(* Logix 5000 project; controller STAT 1756-L72 rev 20.12; software revision 20.04; part 32 of 34 *)
(* tags used below, declared in another part *)
   B3 : DINT[50];
   F8 : REAL[200];
   I2_000_Bit12 : ALIAS FOR stock:2:I.Point_12;   // chaudière wanson0= on 1= off
   I2_000_Bit13 : ALIAS FOR stock:2:I.Point_13;   // chaudière colmatageLigne 30= on 1= off
   I2_001_Bit00 : ALIAS FOR stock:2:I.Point_16;   // NAOHL1 VA4FC O
   I2_001_Bit01 : ALIAS FOR stock:2:I.Point_17;   // NAOHL1 VA4FC F
   I2_001_Bit02 : ALIAS FOR stock:2:I.Point_18;   // NAOHL2 VA4FC O
   I2_001_Bit03 : ALIAS FOR stock:2:I.Point_19;   // NAOHL2 VA4FC O
   I2_001_Bit06 : ALIAS FOR stock:2:I.Point_22;   // pulse debitmetreacide 0.2 l
   I2_001_Bit07 : ALIAS FOR stock:2:I.Point_23;   // pulse eau in tourL1 &2
   I2_001_Bit15 : ALIAS FOR stock:2:I.Point_31;   // pulse 0.1L passé
   I5_000 : ALIAS FOR stock:5:I.Channel_0_Data;
   N20 : DINT[100];
   N7 : DINT[255];
   O3_000_Bit02 : ALIAS FOR stock:3:O.Point_2;   // pompe acide
   O3_000_Bit08 : ALIAS FOR stock:3:O.Point_8;   // vanne soude
   S_V_NAOH : BOOL;
   T4 : TIMER[50];
   dmd_h2so4_ibt_ok : BOOL;
   dmd_soude_ibt_ok : BOOL;
   h2so4_ibt_finit : BOOL;
   ibt_level_soude_plein : BOOL;
   L1_stat : DINT[20];
   L2_STAT : DINT[20];
   L3_STAT : DINT[20];
   lancystock2 : DINT;
   N : INT[255];
   N12 : DINT[230];
   ons12 : BOOL;
   ONS13 : BOOL;
   ONS3 : BOOL;
   ONS4 : BOOL;
   ONS5 : BOOL;
   s_acide_ibt_passe : REAL;
   s_bp_start_h2so4_ibt : BOOL;
   s_bp_stop_acide_ibt : BOOL;
   s_bp_stop_soude_ibt : BOOL;
   s_dmd_acid_ibt : DINT;
   s_h2so4_ibt : BOOL;
   S_naoh_ibt : BOOL;
   S_naoh_ibt_passe : REAL;
   S_stock_v_h2so4_f : BOOL;
   S_stock_v_h2so4_o : BOOL;
   S_stock_v_naoh_o : BOOL;
   stat_L1 : DINT[20];
   STAT_L2 : DINT[20];
   STAT_L3 : DINT[20];
   stocklancy1 : DINT;
   stocklancy2 : DINT;
   stocklancy3 : DINT;
   tot_gaz_chaud_iwts_L123 : DINT;   // 19/1/15 13h45
   tot_gaz_chaud_L3 : DINT;   // debut le 16/1/15 à 11h30
   tot_gaz_chaud_wanson : DINT;   // 19/1/15 13h45
   tot_h2so4_stat : REAL;
(* stock, continued *)

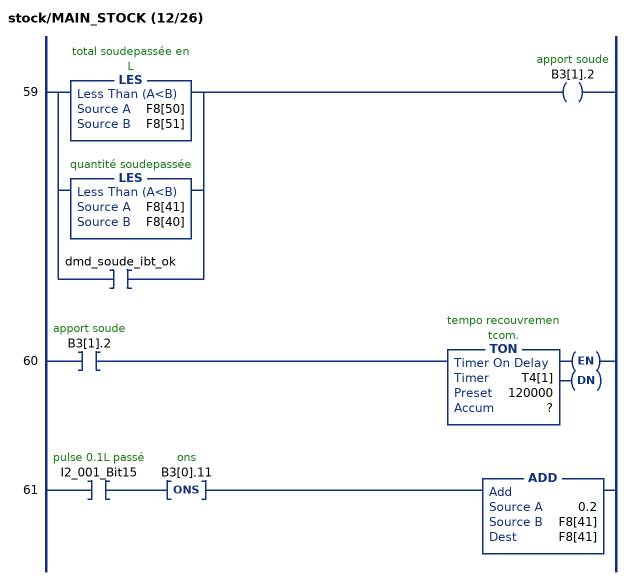
   [picture p650: stock/MAIN_STOCK rungs 59-61]
   59: [LES(F8[50],F8[51]) ,LES(F8[41],F8[40]) ,XIC(dmd_soude_ibt_ok) ]OTE(B3[1].2);
   60: XIC(B3[1].2)TON(T4[1],?,?);
   61: XIC(I2_001_Bit15)ONS(B3[0].11)ADD(0.2,F8[41],F8[41]);
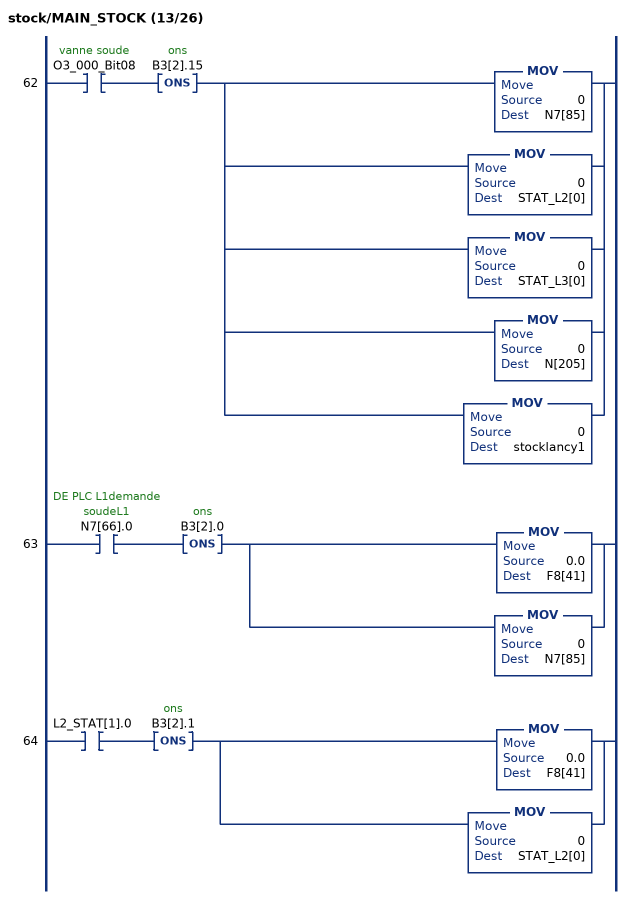
   62: XIC(O3_000_Bit08)ONS(B3[2].15)[MOV(0,N7[85]) ,MOV(0,STAT_L2[0]) ,MOV(0,STAT_L3[0]) ,MOV(0,N[205]) ,MOV(0,stocklancy1) ];
   63: XIC(N7[66].0)ONS(B3[2].0)[MOV(0.0,F8[41]) ,MOV(0,N7[85]) ];
   64: XIC(L2_STAT[1].0)ONS(B3[2].1)[MOV(0.0,F8[41]) ,MOV(0,STAT_L2[0]) ];
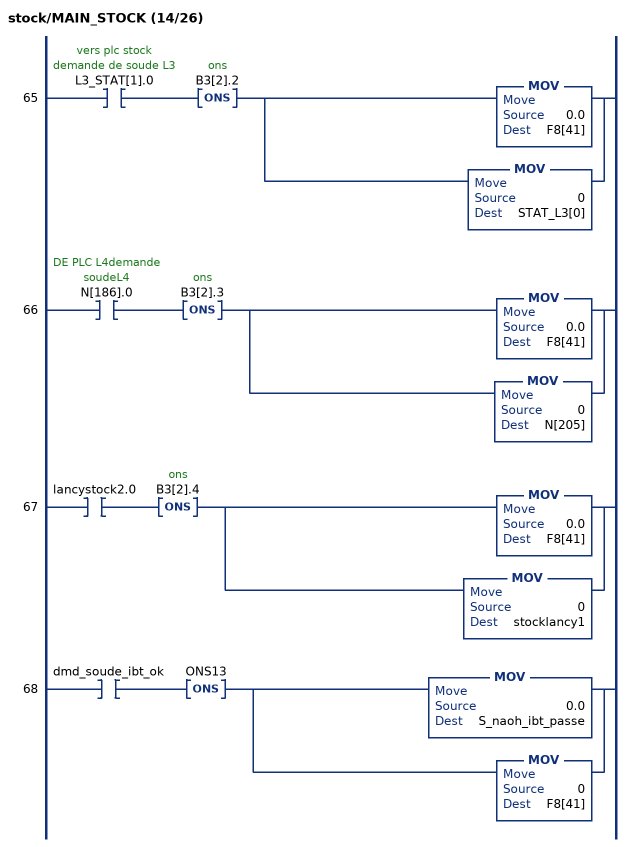
   65: XIC(L3_STAT[1].0)ONS(B3[2].2)[MOV(0.0,F8[41]) ,MOV(0,STAT_L3[0]) ];
   66: XIC(N[186].0)ONS(B3[2].3)[MOV(0.0,F8[41]) ,MOV(0,N[205]) ];
   67: XIC(lancystock2.0)ONS(B3[2].4)[MOV(0.0,F8[41]) ,MOV(0,stocklancy1) ];
   68: XIC(dmd_soude_ibt_ok)ONS(ONS13)[MOV(0.0,S_naoh_ibt_passe) ,MOV(0,F8[41]) ];
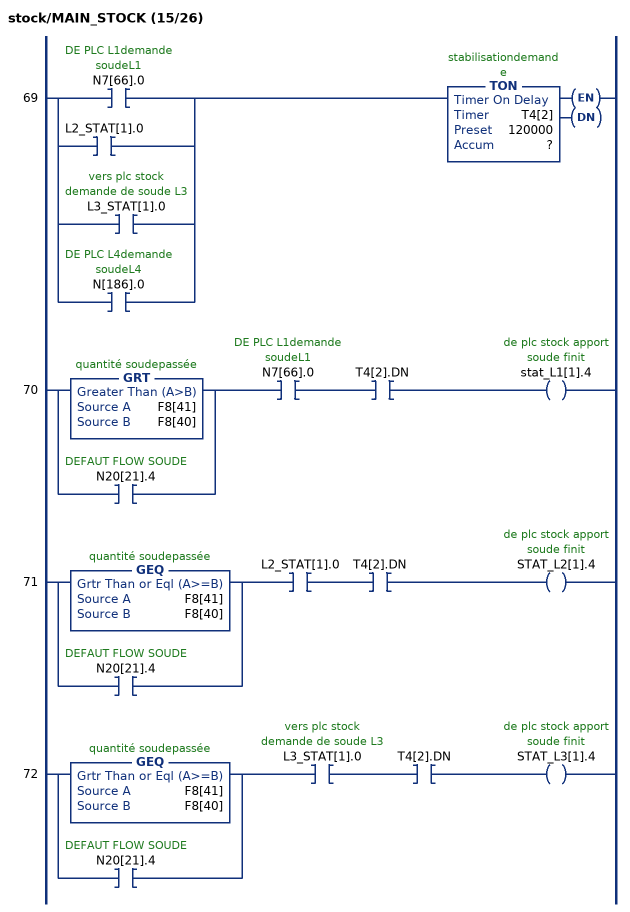
   69: [XIC(N7[66].0) ,XIC(L2_STAT[1].0) ,XIC(L3_STAT[1].0) ,XIC(N[186].0) ]TON(T4[2],?,?);
   70: [GRT(F8[41],F8[40]) ,XIC(N20[21].4) ]XIC(N7[66].0)XIC(T4[2].DN)OTE(stat_L1[1].4);
   71: [GEQ(F8[41],F8[40]) ,XIC(N20[21].4) ]XIC(L2_STAT[1].0)XIC(T4[2].DN)OTE(STAT_L2[1].4);
   72: [GEQ(F8[41],F8[40]) ,XIC(N20[21].4) ]XIC(L3_STAT[1].0)XIC(T4[2].DN)OTE(STAT_L3[1].4);
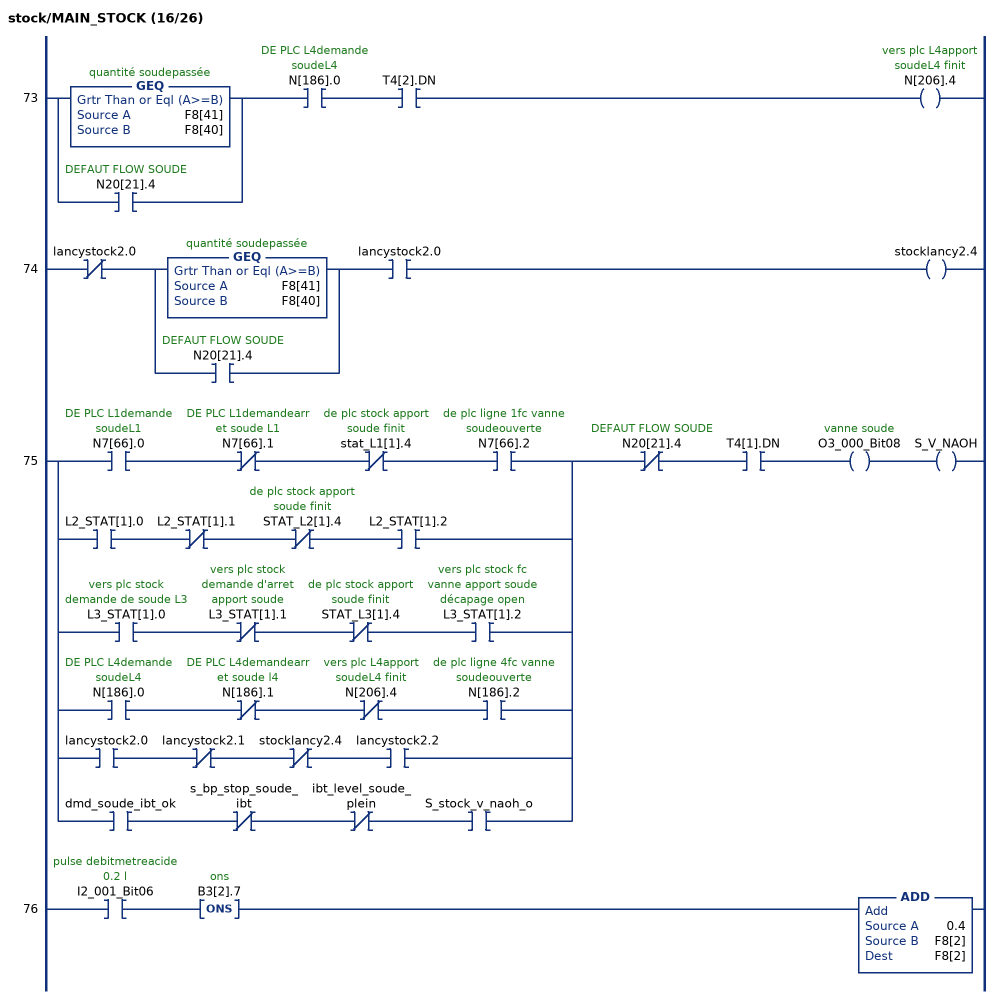
   73: [GEQ(F8[41],F8[40]) ,XIC(N20[21].4) ]XIC(N[186].0)XIC(T4[2].DN)OTE(N[206].4);
   74: XIO(lancystock2.0)[GEQ(F8[41],F8[40]) ,XIC(N20[21].4) ]XIC(lancystock2.0)OTE(stocklancy2.4);
   75: [XIC(N7[66].0) XIO(N7[66].1) XIO(stat_L1[1].4) XIC(N7[66].2) ,XIC(L2_STAT[1].0) XIO(L2_STAT[1].1) XIO(STAT_L2[1].4) XIC(L2_STAT[1].2) ,XIC(L3_STAT[1].0) XIO(L3_STAT[1].1) XIO(STAT_L3[1].4) XIC(L3_STAT[1].2) ,XIC(N[186].0) XIO(N[186].1) XIO(N[206].4) XIC(N[186].2) ,XIC(lancystock2.0) XIO(lancystock2.1) XIO(stocklancy2.4) XIC(lancystock2.2) ,XIC(dmd_soude_ibt_ok) XIO(s_bp_stop_soude_ibt) XIO(ibt_level_soude_plein) XIC(S_stock_v_naoh_o) ]XIO(N20[21].4)XIC(T4[1].DN)OTE(O3_000_Bit08)OTE(S_V_NAOH);
   76: XIC(I2_001_Bit06)ONS(B3[2].7)ADD(0.4,F8[2],F8[2]);
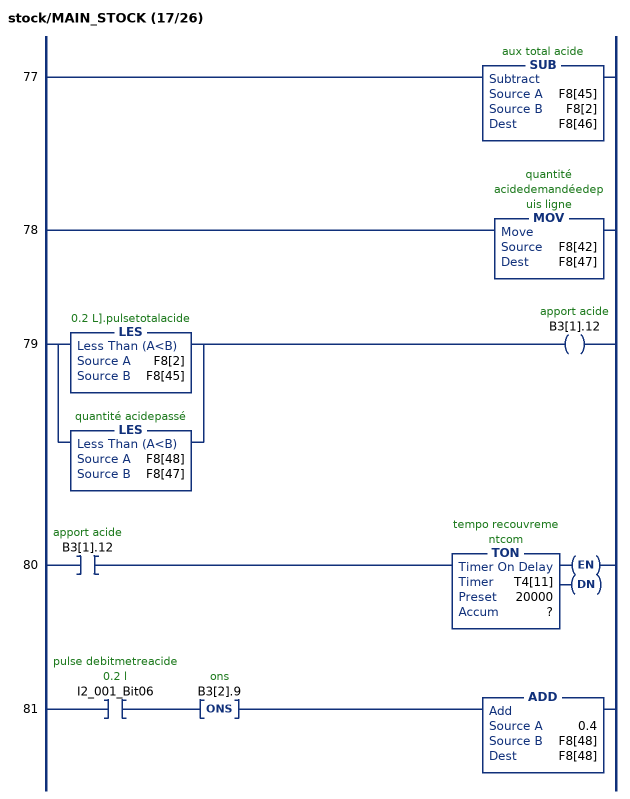
   77: SUB(F8[45],F8[2],F8[46]);
   78: MOV(F8[42],F8[47]);
   79: [LES(F8[2],F8[45]) ,LES(F8[48],F8[47]) ]OTE(B3[1].12);
   80: XIC(B3[1].12)TON(T4[11],?,?);
   81: XIC(I2_001_Bit06)ONS(B3[2].9)ADD(0.4,F8[48],F8[48]);
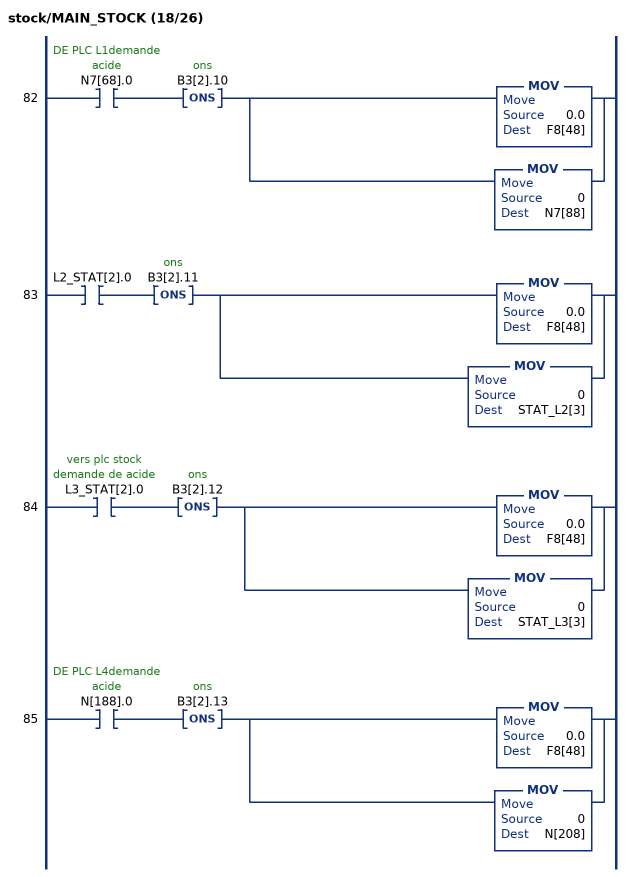
   82: XIC(N7[68].0)ONS(B3[2].10)[MOV(0.0,F8[48]) ,MOV(0,N7[88]) ];
   83: XIC(L2_STAT[2].0)ONS(B3[2].11)[MOV(0.0,F8[48]) ,MOV(0,STAT_L2[3]) ];
   84: XIC(L3_STAT[2].0)ONS(B3[2].12)[MOV(0.0,F8[48]) ,MOV(0,STAT_L3[3]) ];
   85: XIC(N[188].0)ONS(B3[2].13)[MOV(0.0,F8[48]) ,MOV(0,N[208]) ];
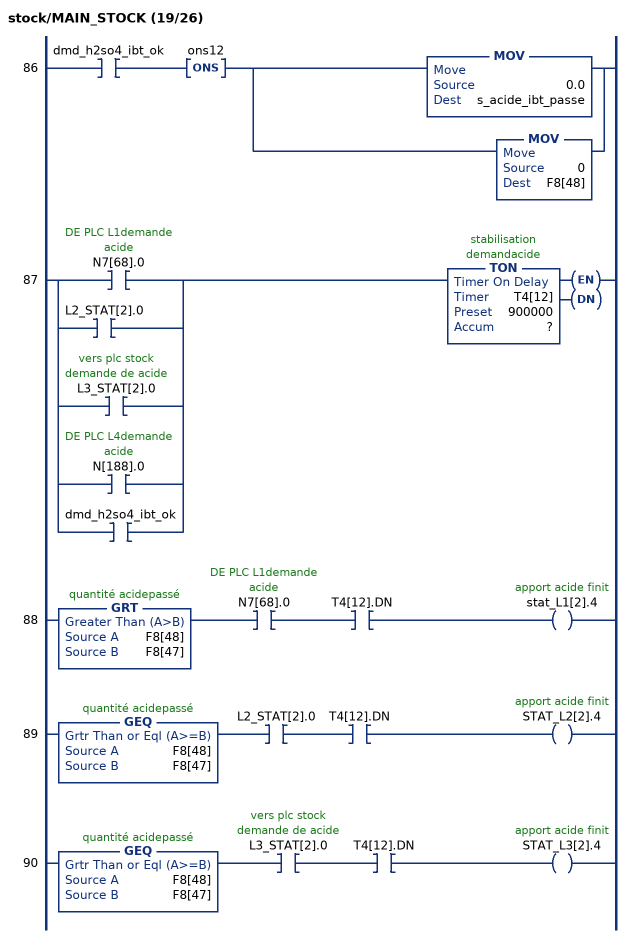
   86: XIC(dmd_h2so4_ibt_ok)ONS(ons12)[MOV(0.0,s_acide_ibt_passe) ,MOV(0,F8[48]) ];
   87: [XIC(N7[68].0) ,XIC(L2_STAT[2].0) ,XIC(L3_STAT[2].0) ,XIC(N[188].0) ,XIC(dmd_h2so4_ibt_ok) ]TON(T4[12],?,?);
   88: GRT(F8[48],F8[47])XIC(N7[68].0)XIC(T4[12].DN)OTE(stat_L1[2].4);
   89: GEQ(F8[48],F8[47])XIC(L2_STAT[2].0)XIC(T4[12].DN)OTE(STAT_L2[2].4);
   90: GEQ(F8[48],F8[47])XIC(L3_STAT[2].0)XIC(T4[12].DN)OTE(STAT_L3[2].4);
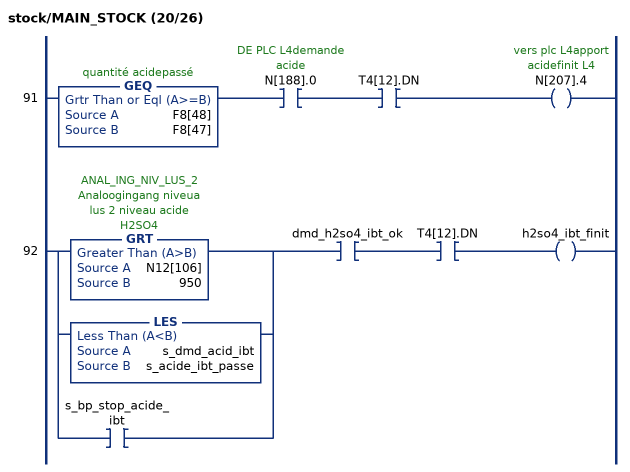
   91: GEQ(F8[48],F8[47])XIC(N[188].0)XIC(T4[12].DN)OTE(N[207].4);
   92: [GRT(N12[106],950) ,LES(s_dmd_acid_ibt,s_acide_ibt_passe) ,XIC(s_bp_stop_acide_ibt) ]XIC(dmd_h2so4_ibt_ok)XIC(T4[12].DN)OTE(h2so4_ibt_finit);
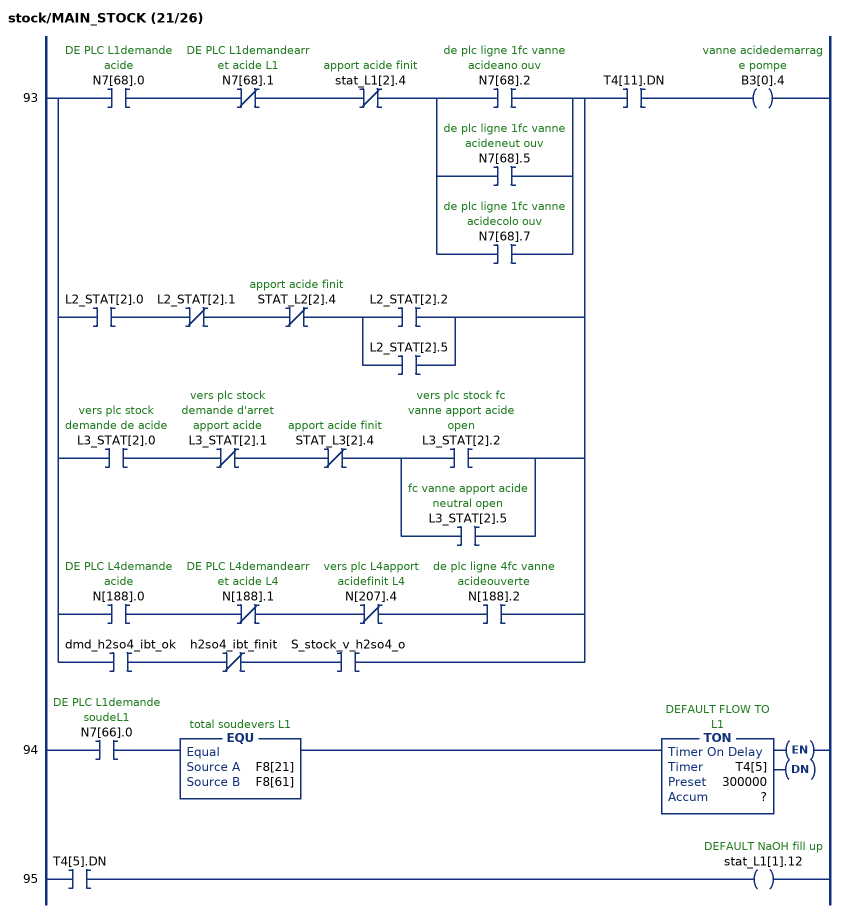
   93: [XIC(N7[68].0) XIO(N7[68].1) XIO(stat_L1[2].4) [XIC(N7[68].2) ,XIC(N7[68].5) ,XIC(N7[68].7) ] ,XIC(L2_STAT[2].0) XIO(L2_STAT[2].1) XIO(STAT_L2[2].4) [XIC(L2_STAT[2].2) ,XIC(L2_STAT[2].5) ] ,XIC(L3_STAT[2].0) XIO(L3_STAT[2].1) XIO(STAT_L3[2].4) [XIC(L3_STAT[2].2) ,XIC(L3_STAT[2].5) ] ,XIC(N[188].0) XIO(N[188].1) XIO(N[207].4) XIC(N[188].2) ,XIC(dmd_h2so4_ibt_ok) XIO(h2so4_ibt_finit) XIC(S_stock_v_h2so4_o) ]XIC(T4[11].DN)OTE(B3[0].4);
   94: XIC(N7[66].0)EQU(F8[21],F8[61])TON(T4[5],?,?);
   95: XIC(T4[5].DN)OTE(stat_L1[1].12);
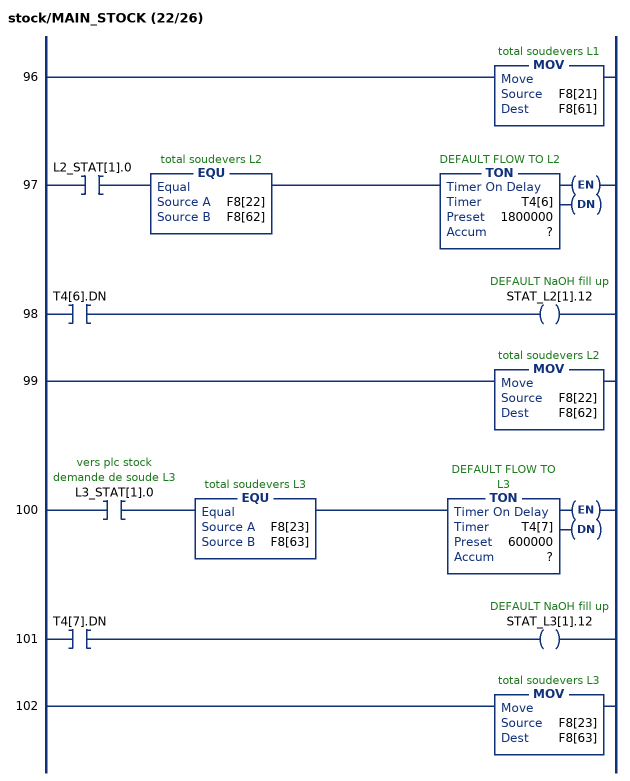
   96: MOV(F8[21],F8[61]);
   97: XIC(L2_STAT[1].0)EQU(F8[22],F8[62])TON(T4[6],?,?);
   98: XIC(T4[6].DN)OTE(STAT_L2[1].12);
   99: MOV(F8[22],F8[62]);
   100: XIC(L3_STAT[1].0)EQU(F8[23],F8[63])TON(T4[7],?,?);
   101: XIC(T4[7].DN)OTE(STAT_L3[1].12);
   102: MOV(F8[23],F8[63]);
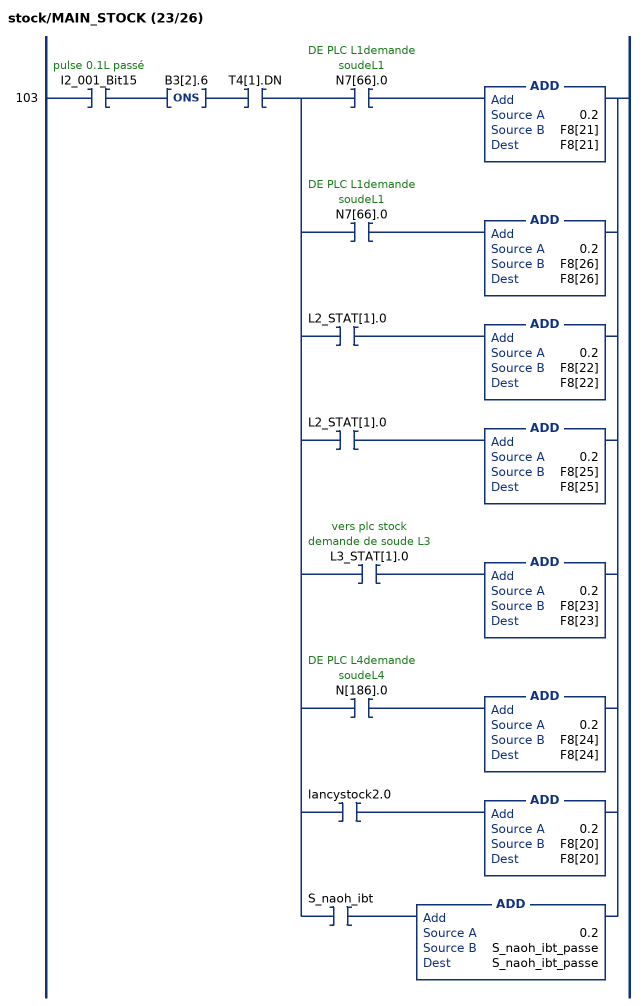
   103: XIC(I2_001_Bit15)ONS(B3[2].6)XIC(T4[1].DN)[XIC(N7[66].0) ADD(0.2,F8[21],F8[21]) ,XIC(N7[66].0) ADD(0.2,F8[26],F8[26]) ,XIC(L2_STAT[1].0) ADD(0.2,F8[22],F8[22]) ,XIC(L2_STAT[1].0) ADD(0.2,F8[25],F8[25]) ,XIC(L3_STAT[1].0) ADD(0.2,F8[23],F8[23]) ,XIC(N[186].0) ADD(0.2,F8[24],F8[24]) ,XIC(lancystock2.0) ADD(0.2,F8[20],F8[20]) ,XIC(S_naoh_ibt) ADD(0.2,S_naoh_ibt_passe,S_naoh_ibt_passe) ];
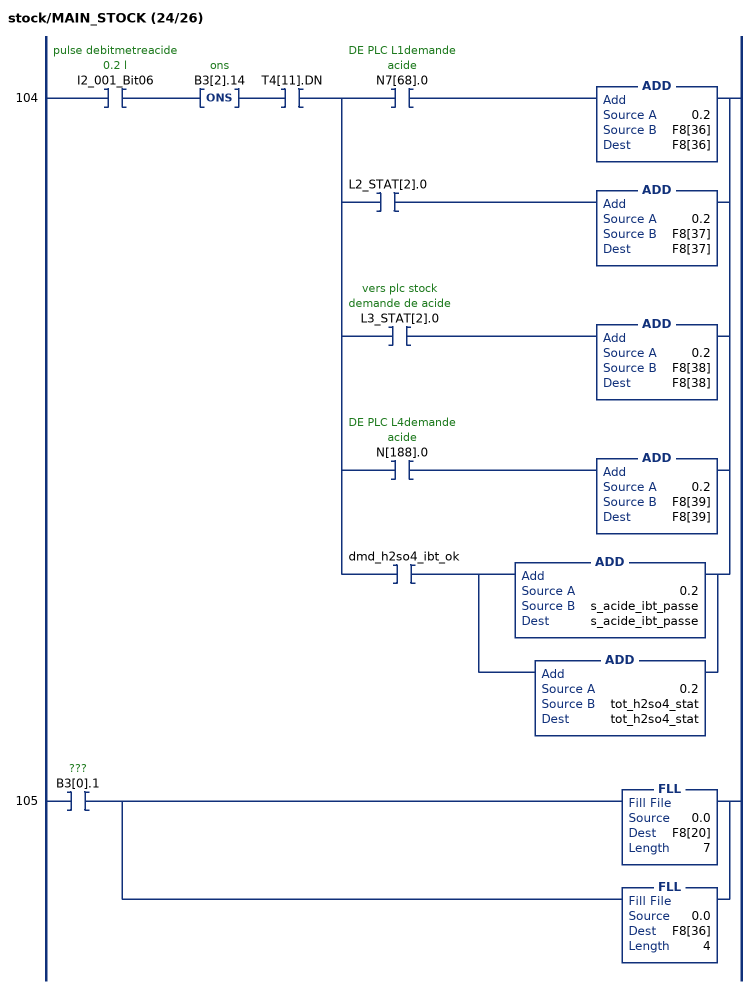
   104: XIC(I2_001_Bit06)ONS(B3[2].14)XIC(T4[11].DN)[XIC(N7[68].0) ADD(0.2,F8[36],F8[36]) ,XIC(L2_STAT[2].0) ADD(0.2,F8[37],F8[37]) ,XIC(L3_STAT[2].0) ADD(0.2,F8[38],F8[38]) ,XIC(N[188].0) ADD(0.2,F8[39],F8[39]) ,XIC(dmd_h2so4_ibt_ok) [ADD(0.2,s_acide_ibt_passe,s_acide_ibt_passe) ,ADD(0.2,tot_h2so4_stat,tot_h2so4_stat) ] ];
   105: XIC(B3[0].1)[FLL(0.0,F8[20],7) ,FLL(0.0,F8[36],4) ];
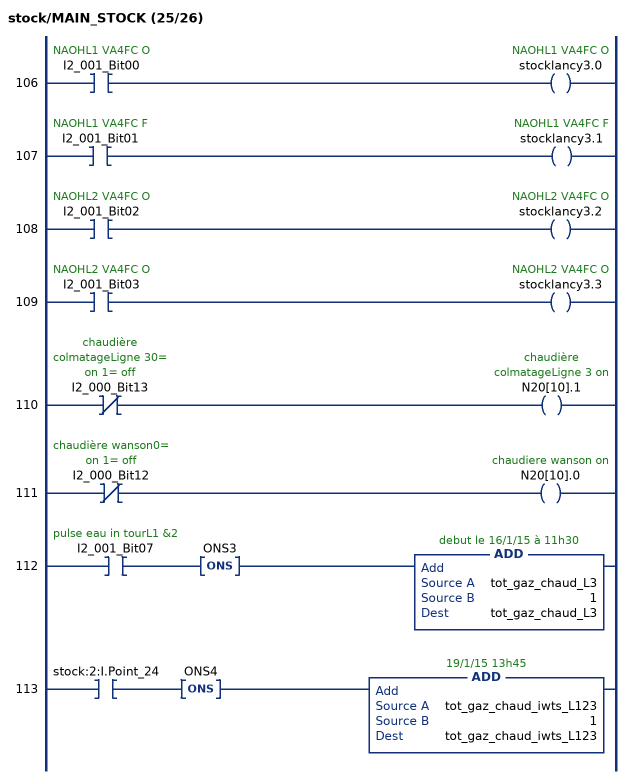
   106: XIC(I2_001_Bit00)OTE(stocklancy3.0);
   107: XIC(I2_001_Bit01)OTE(stocklancy3.1);
   108: XIC(I2_001_Bit02)OTE(stocklancy3.2);
   109: XIC(I2_001_Bit03)OTE(stocklancy3.3);
   110: XIO(I2_000_Bit13)OTE(N20[10].1);
   111: XIO(I2_000_Bit12)OTE(N20[10].0);
   112: XIC(I2_001_Bit07)ONS(ONS3)ADD(tot_gaz_chaud_L3,1,tot_gaz_chaud_L3);
   113: XIC(stock:2:I.Point_24)ONS(ONS4)ADD(tot_gaz_chaud_iwts_L123,1,tot_gaz_chaud_iwts_L123);
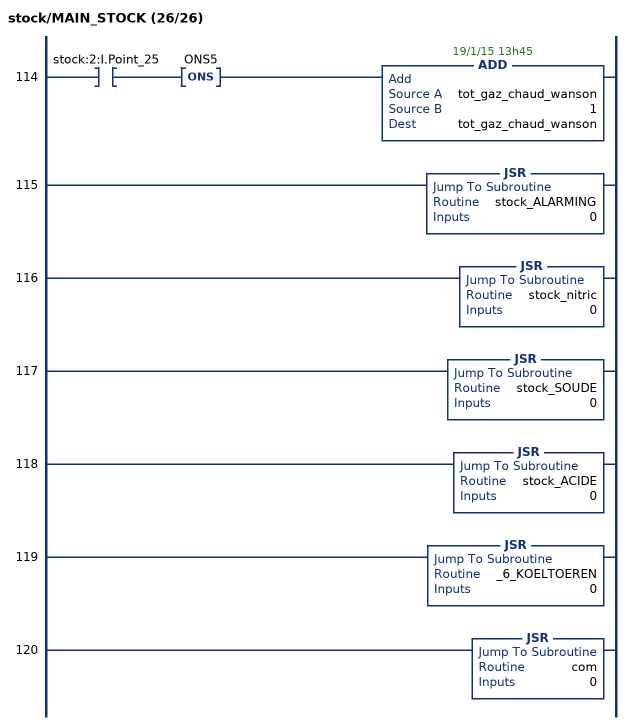
   114: XIC(stock:2:I.Point_25)ONS(ONS5)ADD(tot_gaz_chaud_wanson,1,tot_gaz_chaud_wanson);
   115: JSR(stock_ALARMING,0);
   116: JSR(stock_nitric,0);
   117: JSR(stock_SOUDE,0);
   118: JSR(stock_ACIDE,0);
   119: JSR(_6_KOELTOEREN,0);
   120: JSR(com,0);
END_ROUTINE

ROUTINE stock_ACIDE   (* ladder *)
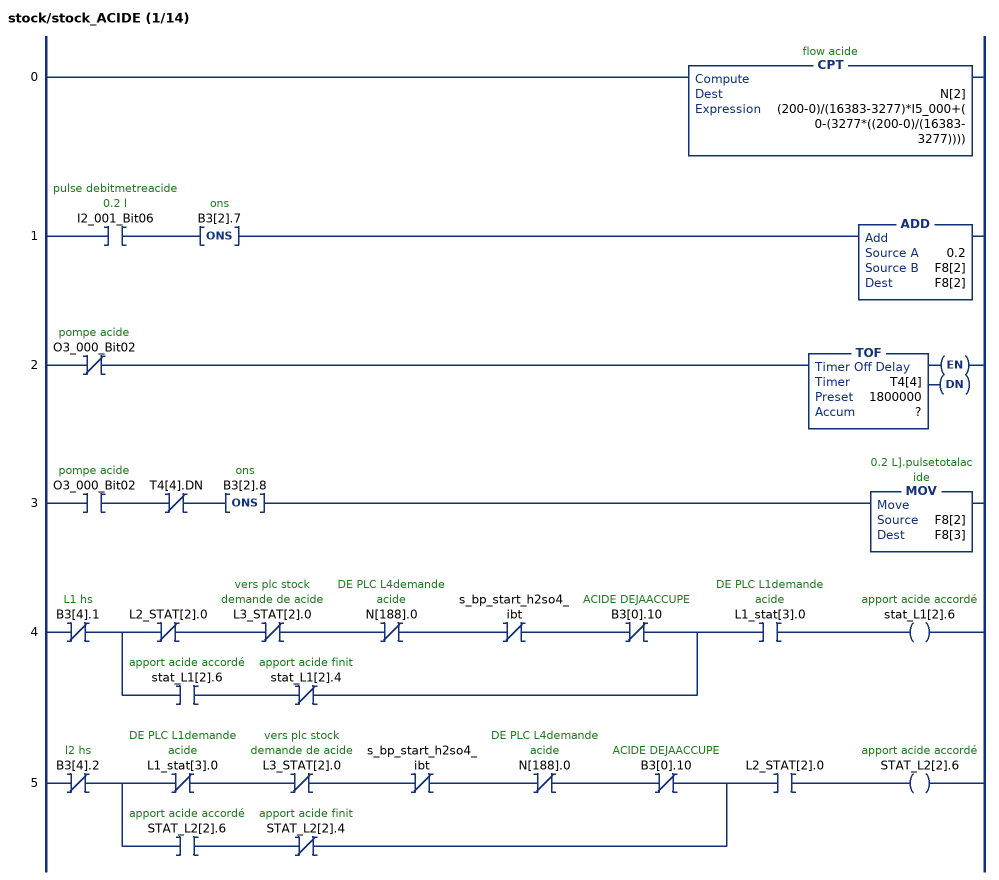
   0: CPT(N[2],(200-0)/(16383-3277)*I5_000+(0-(3277*((200-0)/(16383-3277)))));
   1: XIC(I2_001_Bit06)ONS(B3[2].7)ADD(0.2,F8[2],F8[2]);
   2: XIO(O3_000_Bit02)TOF(T4[4],?,?);
   3: XIC(O3_000_Bit02)XIO(T4[4].DN)ONS(B3[2].8)MOV(F8[2],F8[3]);
   4: XIO(B3[4].1)[XIO(L2_STAT[2].0) XIO(L3_STAT[2].0) XIO(N[188].0) XIO(s_bp_start_h2so4_ibt) XIO(B3[0].10) ,XIC(stat_L1[2].6) XIO(stat_L1[2].4) ]XIC(L1_stat[3].0)OTE(stat_L1[2].6);
   5: XIO(B3[4].2)[XIO(L1_stat[3].0) XIO(L3_STAT[2].0) XIO(s_bp_start_h2so4_ibt) XIO(N[188].0) XIO(B3[0].10) ,XIC(STAT_L2[2].6) XIO(STAT_L2[2].4) ]XIC(L2_STAT[2].0)OTE(STAT_L2[2].6);
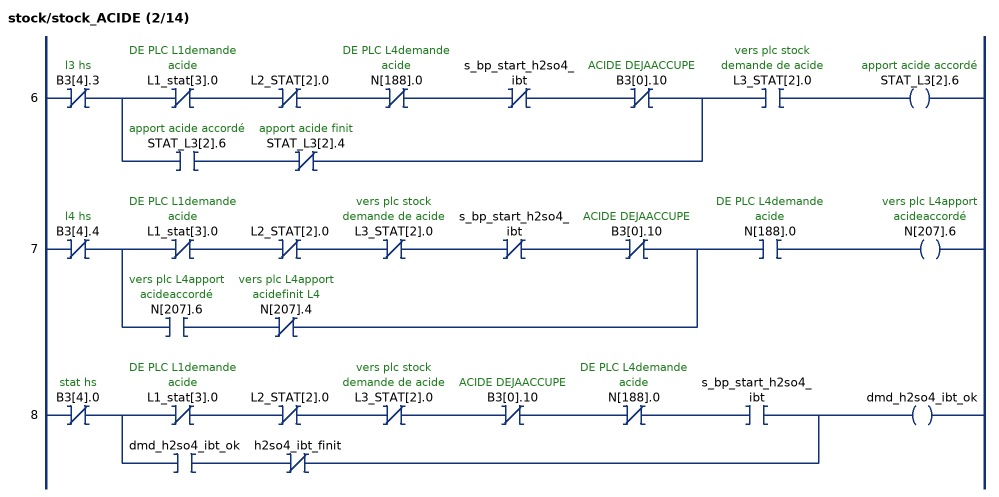
   6: XIO(B3[4].3)[XIO(L1_stat[3].0) XIO(L2_STAT[2].0) XIO(N[188].0) XIO(s_bp_start_h2so4_ibt) XIO(B3[0].10) ,XIC(STAT_L3[2].6) XIO(STAT_L3[2].4) ]XIC(L3_STAT[2].0)OTE(STAT_L3[2].6);
   7: XIO(B3[4].4)[XIO(L1_stat[3].0) XIO(L2_STAT[2].0) XIO(L3_STAT[2].0) XIO(s_bp_start_h2so4_ibt) XIO(B3[0].10) ,XIC(N[207].6) XIO(N[207].4) ]XIC(N[188].0)OTE(N[207].6);
   8: XIO(B3[4].0)[XIO(L1_stat[3].0) XIO(L2_STAT[2].0) XIO(L3_STAT[2].0) XIO(B3[0].10) XIO(N[188].0) XIC(s_bp_start_h2so4_ibt) ,XIC(dmd_h2so4_ibt_ok) XIO(h2so4_ibt_finit) ]OTE(dmd_h2so4_ibt_ok);
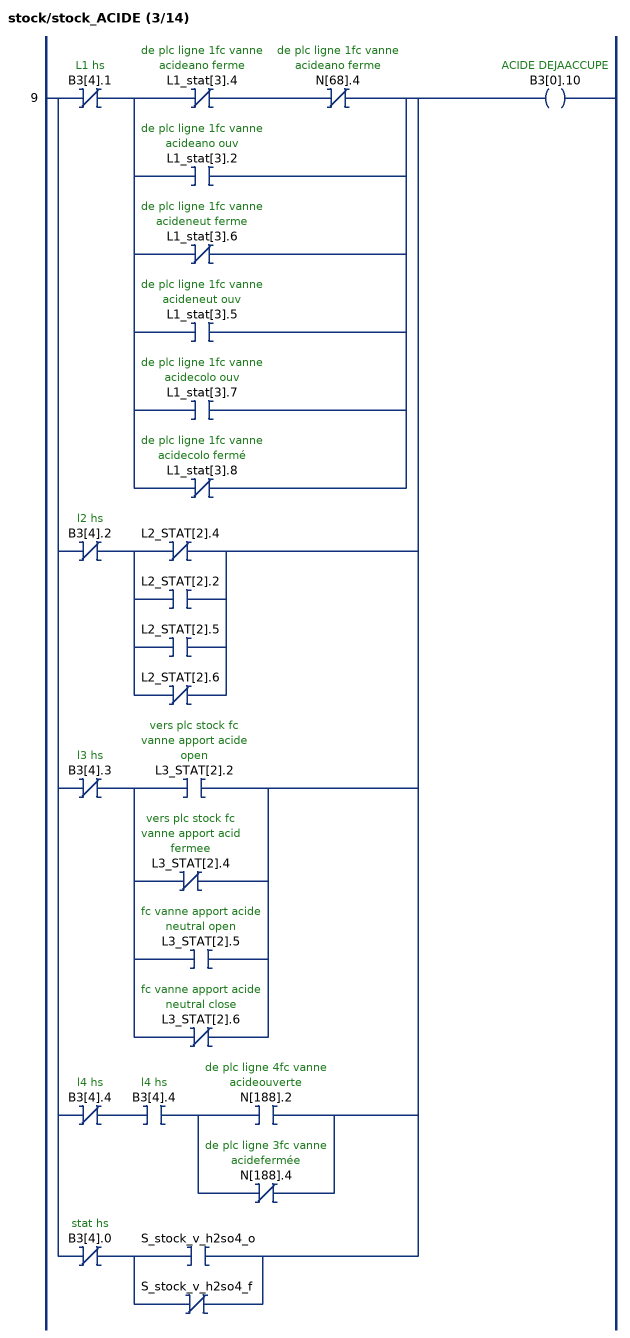
   9: [XIO(B3[4].1) [XIO(L1_stat[3].4) XIO(N[68].4) ,XIC(L1_stat[3].2) ,XIO(L1_stat[3].6) ,XIC(L1_stat[3].5) ,XIC(L1_stat[3].7) ,XIO(L1_stat[3].8) ] ,XIO(B3[4].2) [XIO(L2_STAT[2].4) ,XIC(L2_STAT[2].2) ,XIC(L2_STAT[2].5) ,XIO(L2_STAT[2].6) ] ,XIO(B3[4].3) [XIC(L3_STAT[2].2) ,XIO(L3_STAT[2].4) ,XIC(L3_STAT[2].5) ,XIO(L3_STAT[2].6) ] ,XIO(B3[4].4) XIC(B3[4].4) [XIC(N[188].2) ,XIO(N[188].4) ] ,XIO(B3[4].0) [XIC(S_stock_v_h2so4_o) ,XIO(S_stock_v_h2so4_f) ] ]OTE(B3[0].10);
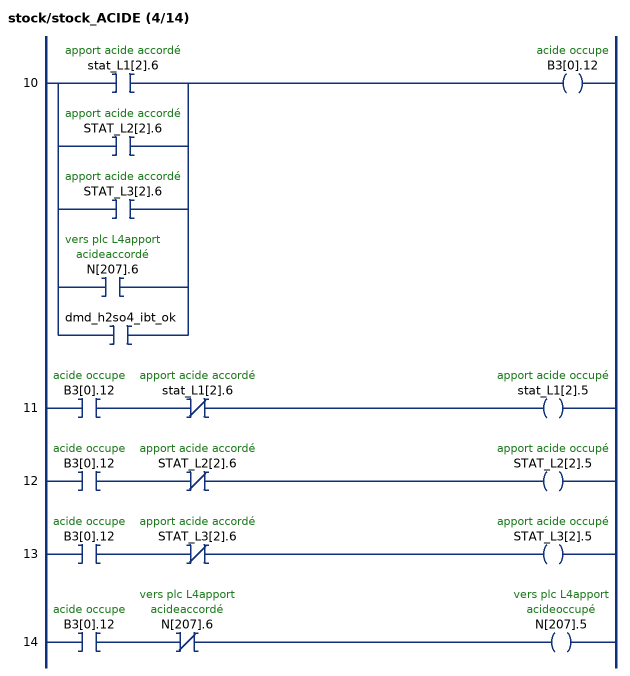
   10: [XIC(stat_L1[2].6) ,XIC(STAT_L2[2].6) ,XIC(STAT_L3[2].6) ,XIC(N[207].6) ,XIC(dmd_h2so4_ibt_ok) ]OTE(B3[0].12);
   11: XIC(B3[0].12)XIO(stat_L1[2].6)OTE(stat_L1[2].5);
   12: XIC(B3[0].12)XIO(STAT_L2[2].6)OTE(STAT_L2[2].5);
   13: XIC(B3[0].12)XIO(STAT_L3[2].6)OTE(STAT_L3[2].5);
   14: XIC(B3[0].12)XIO(N[207].6)OTE(N[207].5);
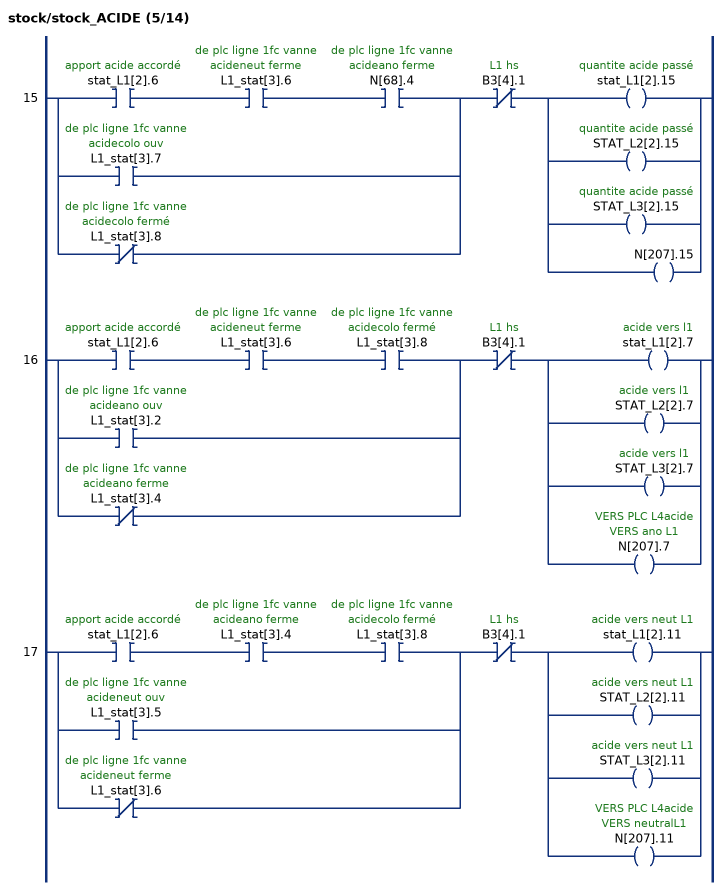
   15: [XIC(stat_L1[2].6) XIC(L1_stat[3].6) XIC(N[68].4) ,XIC(L1_stat[3].7) ,XIO(L1_stat[3].8) ]XIO(B3[4].1)[OTE(stat_L1[2].15) ,OTE(STAT_L2[2].15) ,OTE(STAT_L3[2].15) ,OTE(N[207].15) ];
   16: [XIC(stat_L1[2].6) XIC(L1_stat[3].6) XIC(L1_stat[3].8) ,XIC(L1_stat[3].2) ,XIO(L1_stat[3].4) ]XIO(B3[4].1)[OTE(stat_L1[2].7) ,OTE(STAT_L2[2].7) ,OTE(STAT_L3[2].7) ,OTE(N[207].7) ];
   17: [XIC(stat_L1[2].6) XIC(L1_stat[3].4) XIC(L1_stat[3].8) ,XIC(L1_stat[3].5) ,XIO(L1_stat[3].6) ]XIO(B3[4].1)[OTE(stat_L1[2].11) ,OTE(STAT_L2[2].11) ,OTE(STAT_L3[2].11) ,OTE(N[207].11) ];
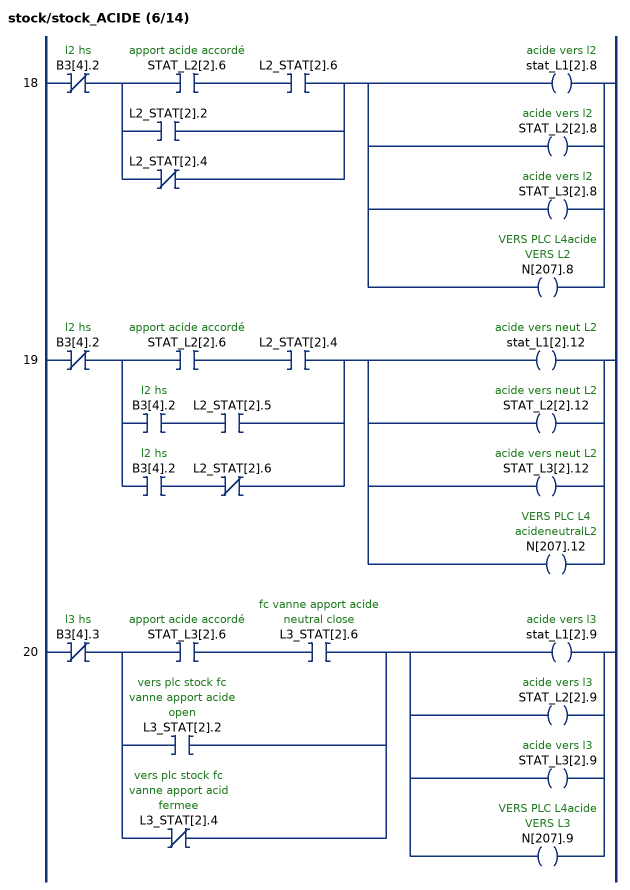
   18: XIO(B3[4].2)[XIC(STAT_L2[2].6) XIC(L2_STAT[2].6) ,XIC(L2_STAT[2].2) ,XIO(L2_STAT[2].4) ][OTE(stat_L1[2].8) ,OTE(STAT_L2[2].8) ,OTE(STAT_L3[2].8) ,OTE(N[207].8) ];
   19: XIO(B3[4].2)[XIC(STAT_L2[2].6) XIC(L2_STAT[2].4) ,XIC(B3[4].2) XIC(L2_STAT[2].5) ,XIC(B3[4].2) XIO(L2_STAT[2].6) ][OTE(stat_L1[2].12) ,OTE(STAT_L2[2].12) ,OTE(STAT_L3[2].12) ,OTE(N[207].12) ];
   20: XIO(B3[4].3)[XIC(STAT_L3[2].6) XIC(L3_STAT[2].6) ,XIC(L3_STAT[2].2) ,XIO(L3_STAT[2].4) ][OTE(stat_L1[2].9) ,OTE(STAT_L2[2].9) ,OTE(STAT_L3[2].9) ,OTE(N[207].9) ];
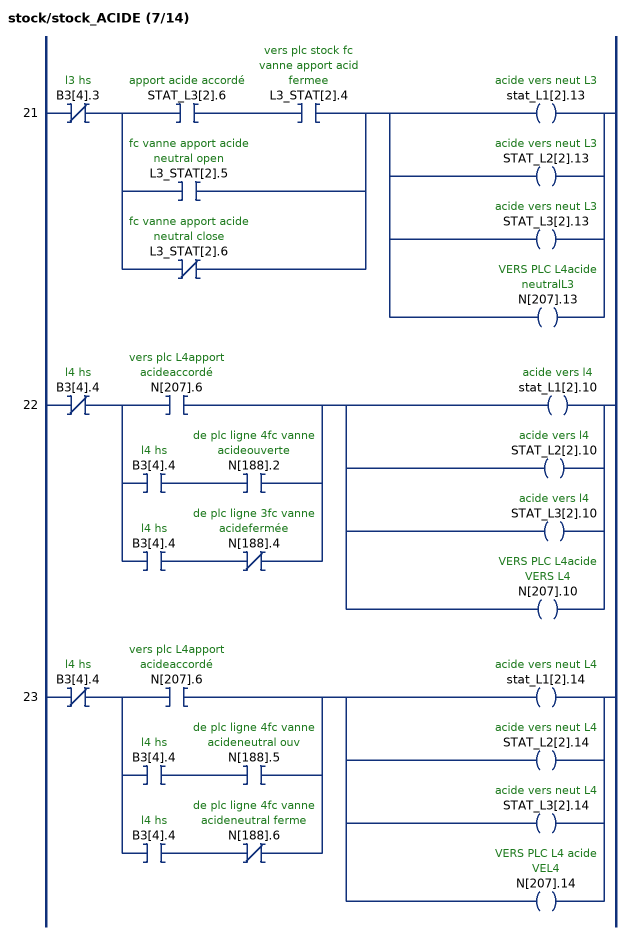
   21: XIO(B3[4].3)[XIC(STAT_L3[2].6) XIC(L3_STAT[2].4) ,XIC(L3_STAT[2].5) ,XIO(L3_STAT[2].6) ][OTE(stat_L1[2].13) ,OTE(STAT_L2[2].13) ,OTE(STAT_L3[2].13) ,OTE(N[207].13) ];
   22: XIO(B3[4].4)[XIC(N[207].6) ,XIC(B3[4].4) XIC(N[188].2) ,XIC(B3[4].4) XIO(N[188].4) ][OTE(stat_L1[2].10) ,OTE(STAT_L2[2].10) ,OTE(STAT_L3[2].10) ,OTE(N[207].10) ];
   23: XIO(B3[4].4)[XIC(N[207].6) ,XIC(B3[4].4) XIC(N[188].5) ,XIC(B3[4].4) XIO(N[188].6) ][OTE(stat_L1[2].14) ,OTE(STAT_L2[2].14) ,OTE(STAT_L3[2].14) ,OTE(N[207].14) ];
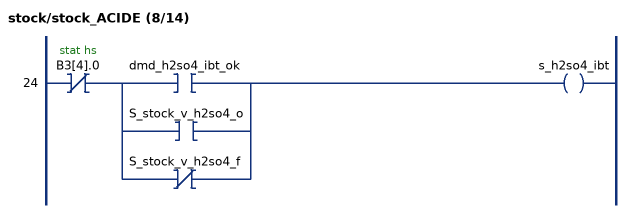
   24: XIO(B3[4].0)[XIC(dmd_h2so4_ibt_ok) ,XIC(S_stock_v_h2so4_o) ,XIO(S_stock_v_h2so4_f) ]OTE(s_h2so4_ibt);
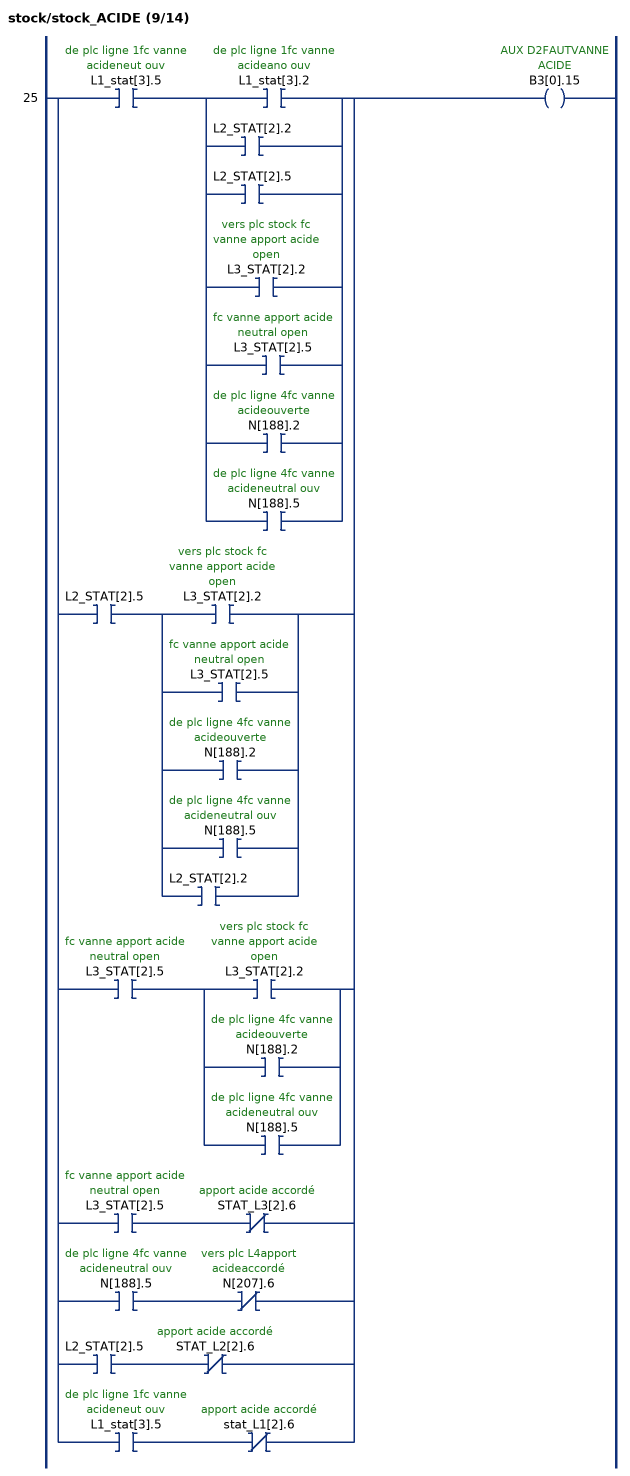
   25: [XIC(L1_stat[3].5) [XIC(L1_stat[3].2) ,XIC(L2_STAT[2].2) ,XIC(L2_STAT[2].5) ,XIC(L3_STAT[2].2) ,XIC(L3_STAT[2].5) ,XIC(N[188].2) ,XIC(N[188].5) ] ,XIC(L2_STAT[2].5) [XIC(L3_STAT[2].2) ,XIC(L3_STAT[2].5) ,XIC(N[188].2) ,XIC(N[188].5) ,XIC(L2_STAT[2].2) ] ,XIC(L3_STAT[2].5) [XIC(L3_STAT[2].2) ,XIC(N[188].2) ,XIC(N[188].5) ] ,XIC(L3_STAT[2].5) XIO(STAT_L3[2].6) ,XIC(N[188].5) XIO(N[207].6) ,XIC(L2_STAT[2].5) XIO(STAT_L2[2].6) ,XIC(L1_stat[3].5) XIO(stat_L1[2].6) ]OTE(B3[0].15);
